// TIA Portal V15.1 export
// export: Created 2024-06-21T08:40:45.8379833Z, ExportSetting WithDefaults, DisplayName Totally Integrated Automation Portal, DisplayVersion V15.1 Update 5, DisplayName TIA Portal Openness, DisplayVersion V15.1 Update 5, DisplayName SINAMICS Startdrive Advanced, DisplayVersion V15.1, DisplayName G130, G150, S120, S150, SINAMICS MV, S210, DisplayVersion V15.1, DisplayName G110M, G120, G120C, G120D, G120P, DisplayVersion V15.1, DisplayName STEP 7 Professional, DisplayVersion V15.1 Update 5, DisplayName STEP 7 Safety, DisplayVersion V15.1, DisplayName WinCC Professional, DisplayVersion V15.1 Update 5, DisplayName SIMATIC Visualization Architect, DisplayVersion V15.1
DATA_BLOCK "_209210ZM01Config"   // DB302
{ S7_Optimized_Access := 'FALSE' }
AUTHOR : VCC
VERSION : 0.1
// stored: AutoNumber false, DBAccessibleFromOPCUA true, IsOnlyStoredInLoadMemory false, IsWriteProtectedInAS false
   VAR
      Andon { ExternalAccessible := 'False'; ExternalVisible := 'False'; ExternalWritable := 'False'} : "AndonConfigVCG";   // Config
      "210CS22ProdSpeed" { ExternalAccessible := 'False'; ExternalVisible := 'False'; ExternalWritable := 'False'} : "ProdSpeedConfig";   // Config
      "210CS22ProdStartStop" { ExternalAccessible := 'False'; ExternalVisible := 'False'; ExternalWritable := 'False'} : "ProdStartStopConfig";   // Config
      "210CS22LineFeed" { ExternalAccessible := 'False'; ExternalVisible := 'False'; ExternalWritable := 'False'} : "LineFeedConfig";   // Config
      "210CS22ShiftRegLine" { ExternalAccessible := 'False'; ExternalVisible := 'False'; ExternalWritable := 'False'} : "ShiftRegLineConfig";   // Config
      "210CHB21" { ExternalAccessible := 'False'; ExternalVisible := 'False'; ExternalWritable := 'False'} : "MovUnit2Pos2S-MoviFitFCPNConfig";   // Config
      "210CR21" { ExternalAccessible := 'False'; ExternalVisible := 'False'; ExternalWritable := 'False'} : "RollerConvMDXPNConfig";   // Config
      "210CS22" { ExternalAccessible := 'False'; ExternalVisible := 'False'; ExternalWritable := 'False'} : "LineConvBrake-MDXPNConfig";   // Config
      "210CR23" { ExternalAccessible := 'False'; ExternalVisible := 'False'; ExternalWritable := 'False'} : "RollerConvMDXPNConfig";   // Config
      "210ASH01" { ExternalAccessible := 'False'; ExternalVisible := 'False'; ExternalWritable := 'False'} : "HandHeldHBA-Config";   // Config
   END_VAR
BEGIN
END_DATA_BLOCK
